FUNCTION_BLOCK FB_Machine
VAR_INPUT
	// ========================== SEPARATING MODULE =======================================
	// Separating module - clamp cylinder
	bSeparatingClampDiag						:		BOOL	:=	FALSE;
	bSeparatingClampTemp						:		BOOL	:=	TRUE;
	bSeparatingClampRecord						:		BOOL	:=	TRUE;
	// Separating module - barrier cylinder
	bSeparatingBarrierDiag						:		BOOL	:=	TRUE;
	bSeparatingBarrierTemp						:		BOOL	:=	TRUE;
	bSeparatingBarrierRecord					:		BOOL	:=	FALSE;
	// ========================== SORTING MODULES ==========================================
	bMetalSortingCylinderDiag					:		BOOL	:= 	TRUE;
	bMetalSortingCylinderTemp					:		BOOL	:=	FALSE;
	bMetalSortingCylinderRecord					:		BOOL	:=	FALSE;
	
	bPlasticSortingCylinderDiag					:		BOOL	:=	FALSE;
	bPlasticSortingCylinderTemp					:		BOOL	:=	FALSE;
	bPlasticSortingCylinderRecord				:		BOOL	:=	FALSE;
END_VAR
VAR
	// ============================= ERROR ==================================================
	bError										:		BOOL;
	// ========================== Axis Variable =============================================
	fAxisVelo									:		LREAL;
	fAxisVeloLastCycle							:		LREAL;
	// ======================== State machine variables =====================================
	bStarted									:		BOOL;
	bStopped									:		BOOL;
	bReset								AT %Q* 	: 		BOOL;
	bAborted									:		BOOL;
	bIdle										:		BOOL;
	bAuto										:		BOOL;
	bSemi										:		BOOL;
	bManual										:		BOOL;
	bMaintenance								:		BOOL;
	// ========================== Machine submodules ========================================
	fbSeparatingModule							:		FB_SeparatingModule;
	fbMetalSortingModule						:		FB_SortingModule;
	fbPlasticSortingModule						:		FB_SortingModule;
	fbComprAir									:		FB_SignalHandlingIntern;
	fbPowerSupply								:		FB_SignalHandlingIntern;
	// Visualization
	// ========================== Buttons ========================================
	fbButtonStart								:		FB_SignalHandlingIntern;
	fbButtonStop								:		FB_SignalHandlingIntern;
	fbButtonReset								:		FB_SignalHandlingIntern;
	fbButtonAbort								:		FB_SignalHandlingIntern;
	fbButtonAuto								:		FB_SignalHandlingIntern;
	fbButtonSemi								:		FB_SignalHandlingIntern;
	fbButtonManual								:		FB_SignalHandlingIntern;
	fbButtonMaintenance							:		FB_SignalHandlingIntern;
	fbButtonComprAir							:		FB_SignalHandlingIntern;
	fbButtonPower								:		FB_SignalHandlingIntern;
	// ========================== State machine ==================================
	fbStateMachineAuto							:		PS_PackML_StateMachine_Auto;
	fbStateMachineSemiAuto						:		PS_PackML_StateMachine_SemiAuto;
	fbStateMachineManual						:		PS_PackML_StateMachine_Manual;
	fbStateMachineMaintenance					:		PS_PackML_StateMachine_Maintenance;
	
	e_PMLState									:		E_PMLState			:=	E_PMLState.IDLE;
	e_PMLStateRequest							:		E_PMLState;
	e_PMLUnitMode								:		E_PMLUnitMode		:=	E_PMLUnitMode.IDLE;
	e_PMLUnitModeRequest						:		E_PMLUnitMode;
		fbUnitModeManager						:		PS_PackML_UnitModeManager;
	// ======================= Common variables ===================================
	bInit										:		BOOL;
	bAxisEnable									:		BOOL;
	bManualAxisEnable							:		BOOL;
	
	fbTriggerStartButton						:		R_TRIG;
	fbTriggerSeparated							:		R_TRIG;
	fbTriggerMetalSorted						:		R_TRIG;
	fbTriggerPlasticSorted						:		R_TRIG;
	
	nBoxesOnTransport							:		UINT;
	
	aClampTemps									:		ARRAY [1..100] OF LREAL;
	aBarrierTemps								:		ARRAY [1..100] OF LREAL;
	aMetalCylTemps								:		ARRAY [1..100] OF LREAL;
	aPlasticCylTemps							:		ARRAY [1..100] OF LREAL;
	
	bStartingIsSetToTrue						:		BOOL;
	bResetIsSetToTrue							:		BOOL;
	bHaltIsSetToTrue							:		BOOL;
END_VAR
VAR CONSTANT
	// ======================= Axis parameters ===================================
	cAxisVeloAutomatic							:		LREAL	:=		100.0;
	cAxisVeloNonAutomatic						:		LREAL	:=		50.0;
	// =============== Separating module parameters ===============================
	tSeparatingTimeOutClamp						:		TIME	:=		T#4S;
	tSeparatingRecordIntervalClamp				:		TIME	:=		T#1S;
	
	tSeparatingTimeOutBarrier					:		TIME	:=		T#3S;
	tSeparatingRecordIntervalBarrier			:		TIME	:=		T#1S;
	tSeparatingTimeBarrierAtWork				:		TIME	:=		T#3.5S;
	
	rSeparatingClampTempMin						:		LREAL	:=		5.0;
	rSeparatingClampTempMax						:		LREAL	:=		78.0;
	rSeparatingBarrierTempMin					:		LREAL	:= 		2.0;
	rSeparatingBarrierTempMax					:		LREAL	:= 		95.0;
	// =============== Sorting module parameters ==================================
	tSortingMetalTimeOutCyl						:		TIME	:=		T#3S;
	tSortingMetalRecordIntervalCyl				:		TIME	:=		T#1S;
	tSortingMetalSensorDelay					:		TIME	:=		T#2S;
	tSortingMetalMoveAxisDelay					:		TIME	:=		T#3S;

	rSortingMetalCylTempMin						:		LREAL	:= 		2.0;
	rSortingMetalCylTempMax						:		LREAL	:= 		95.0;
	
	tSortingPlasticTimeOutCyl					:		TIME	:=		T#3S;
	tSortingPlasticRecordIntervalCyl			:		TIME	:=		T#1S;
	tSortingPlasticSensorDelay					:		TIME	:=		T#2S;
	tSortingPlasticMoveAxisDelay				:		TIME	:=		T#3S;
	
	rSortingPlasticCylTempMin					:		LREAL	:= 		2.0;
	rSortingPlasticCylTempMax					:		LREAL	:= 		95.0;
END_VAR


	// Modules errors
	bError	:=	fbSeparatingModule.bAxisError OR fbSeparatingModule.bBarrierError OR fbSeparatingModule.bClampError OR
				fbMetalSortingModule.bAxisError OR fbMetalSortingModule.bCylError OR
				fbPlasticSortingModule.bAxisError OR fbPlasticSortingModule.bCylError;
				
	// Axis velocity
	IF (e_PMLUnitMode = E_PMLUnitMode.AUTOMATIC OR e_PMLUnitMode = E_PMLUnitMode.SEMIAUTOMATIC) THEN
		fAxisVelo		:=		cAxisVeloAutomatic;
	ELSE
		fAxisVelo		:=		cAxisVeloNonAutomatic;	
	END_IF
 
	// Separeted and sorted boxes output transfer
	fbTriggerSeparated(		CLK		:=		fbSeparatingModule.bSeparated);
	fbTriggerMetalSorted(	CLK		:=		fbMetalSortingModule.bSorted);
	fbTriggerPlasticSorted(	CLK		:=		fbPlasticSortingModule.bSorted);
	
	// Temperatures of modules
	aBarrierTemps					:=		fbSeparatingModule.aBarrierTemp;
	aClampTemps						:=		fbSeparatingModule.aClampTemp;
	aMetalCylTemps					:=		fbMetalSortingModule.aCylTemps;
	aPlasticCylTemps				:=		fbPlasticSortingModule.aCylTemps;
	
	// Cylinder options of modules
	fbSeparatingModule.CylinderOptions(		bClampDiag			:=				bSeparatingClampDiag,
											bClampTemp			:=				bSeparatingClampTemp,
											bClampRecord		:=				bSeparatingClampRecord,
											bBarrierDiag		:=				bSeparatingBarrierDiag,
											bBarrierTemp		:=				bSeparatingBarrierTemp,
											bBarrierRecord		:=				bSeparatingBarrierRecord);
											
	fbMetalSortingModule.CylinderOptions(	bCylDiag			:=				bMetalSortingCylinderDiag,
											bCylTemp			:=				bMetalSortingCylinderTemp,
											bCylRecord			:=				bMetalSortingCylinderRecord);
											
	fbPlasticSortingModule.CylinderOptions(	bCylDiag			:=				bPlasticSortingCylinderDiag,
											bCylTemp			:=				bPlasticSortingCylinderTemp,
											bCylRecord			:=				bPlasticSortingCylinderRecord);
											
	General_Init();
	
	General_Enable();
	
	General_ModuleInputs();
	
	General_SetOutputs();
	
	General_Requests();
	
	General_StateMachine();

METHOD PRIVATE General_Enable
VAR_INPUT
END_VAR

	// Power supply
	fbPowerSupply.Enable(	bEnable					:=		TRUE);
	fbButtonPower.Enable(	bEnable					:=		TRUE);
	
	
	fbPowerSupply.bInputSignal					:=		fbButtonPower.bOutputSignal;
	
	// Axis control
	IF (e_PMLState	:=	E_PMLState.ABORTED) THEN
		bAxisEnable				:=		FALSE;
	ELSIF fbPowerSupply.bOutputSignal THEN
		bAxisEnable				:=		TRUE;		
	END_IF
	
	bManualAxisEnable	:=	fbPowerSupply.bOutputSignal AND (e_PMLState	:=	E_PMLState.EXECUTE) AND (e_PMLUnitMode = E_PMLUnitMode.MANUAL OR e_PMLUnitMode = E_PMLUnitMode.MAINTENANCE);
	
	// Compressed air control
	IF NOT (e_PMLUnitMode		:=		E_PMLUnitMode.MAINTENANCE) THEN
		fbComprAir				:=		fbPowerSupply.bOutputSignal;
	ELSE
		fbComprAir				:=		fbButtonComprAir;
	END_IF
	
	fbComprAir.Enable(			bEnable		:=		TRUE);
	fbButtonComprAir.Enable(	bEnable		:=		(e_PMLUnitMode = E_PMLUnitMode.MAINTENANCE));
	
	// Separating module 
	fbSeparatingModule.Enable(		bAxisEnable				:=			bAxisEnable,
									bComprAirEnable			:=			fbComprAir.bOutputSignal OR fbButtonComprAir.bOutputSignal,
									bManualAxisEnable		:=			bManualAxisEnable,
									bSensorEnable			:=			TRUE);
								
	// Sorting plastic
	fbPlasticSortingModule.Enable(	bAxisEnable				:=			bAxisEnable,
									bComprAirEnable			:=			fbComprAir.bOutputSignal OR fbButtonComprAir.bOutputSignal,
									bManualAxisEnable		:=			bManualAxisEnable,
									bSensorEnable			:=			TRUE);
	
	// Sorting metal
	fbMetalSortingModule.Enable(	bAxisEnable				:=			bAxisEnable,
									bComprAirEnable			:=			fbComprAir.bOutputSignal OR fbButtonComprAir.bOutputSignal,
									bManualAxisEnable		:=			bManualAxisEnable,
									bSensorEnable			:=			TRUE);
									
	// States
	fbButtonStart.Enable		(	bEnable					:=			NOT bError);
	
	fbButtonStop.Enable			(	bEnable					:=			((e_PMLState = E_PMLState.STOPPING) OR (e_PMLState = E_PMLState.EXECUTE) OR (e_PMLState = E_PMLState.IDLE)));
	
	fbButtonAbort.bInputSignal								:=			fbPowerSupply.bOutputSignal;
	fbButtonAbort.Enable		(	bEnable					:=			((e_PMLState = E_PMLState.ABORTING) OR (e_PMLState = E_PMLState.STOPPING) OR (e_PMLState = E_PMLState.EXECUTE) OR (e_PMLState = E_PMLState.RESETTING)));
	
	fbButtonReset.Enable		(	bEnable					:=			(e_PMLState = E_PMLState.STOPPED)); 
	
	// Unit Modes
	fbButtonAuto.Enable			(	bEnable					:=			((e_PMLState = E_PMLState.IDLE) AND (e_PMLUnitMode <> E_PMLUnitMode.AUTOMATIC)));
	
	fbButtonSemi.Enable			(	bEnable					:=			((e_PMLState = E_PMLState.IDLE) AND (e_PMLUnitMode <> E_PMLUnitMode.SEMIAUTOMATIC)));
	
	fbButtonManual.Enable		(	bEnable					:=			((e_PMLState = E_PMLState.IDLE) AND (e_PMLUnitMode <> E_PMLUnitMode.MANUAL)));
	
	fbButtonMaintenance.Enable	(	bEnable					:=			((e_PMLState = E_PMLState.IDLE) AND (e_PMLUnitMode <> E_PMLUnitMode.MAINTENANCE)));
END_METHOD

METHOD PRIVATE General_Init
VAR_INPUT
END_VAR

	IF NOT bInit THEN
	// ================================ Separating module parameters ==========================================
		// Clamp cylinder
		fbSeparatingModule.tProp_TimeIntervalClamp				:=		tSeparatingRecordIntervalClamp;
		fbSeparatingModule.tProp_TimeOutClamp					:=		tSeparatingTimeOutClamp;
		
		fbSeparatingModule.nProp_TempMaxClamp					:=		rSeparatingClampTempMax;
		fbSeparatingModule.nProp_TempMinClamp					:=		rSeparatingClampTempMin;
				
		// Barrier cylinder
		fbSeparatingModule.tProp_TimeIntervalBarrier			:=		tSeparatingRecordIntervalBarrier;
		fbSeparatingModule.tProp_TimeOutBarrier					:=		tSeparatingTimeOutBarrier;
		
		fbSeparatingModule.tBarrierAtWorkPos					:=		tSeparatingTimeBarrierAtWork;
		
		fbSeparatingModule.nProp_TempMaxBarrier					:=		rSeparatingBarrierTempMax;
		fbSeparatingModule.nProp_TempMinBarrier					:=		rSeparatingBarrierTempMin;
	

	// ============================== Sorting metal module parameters ==========================================
		fbMetalSortingModule.tProp_AxisMoving					:=		tSortingMetalMoveAxisDelay;
		fbMetalSortingModule.tProp_CylRecInterval				:=		tSortingMetalRecordIntervalCyl;
		fbMetalSortingModule.tProp_CylTimeOut					:=		tSortingMetalTimeOutCyl;
		fbMetalSortingModule.tProp_SensorDelay					:=		tSortingMetalSensorDelay;
		
		fbMetalSortingModule.nProp_CylTempMax					:=		rSortingMetalCylTempMax;
		fbMetalSortingModule.nProp_CylTempMin					:=		rSortingMetalCylTempMin;
			
	// ============================== Sorting plastic module parameters ==========================================
		fbPlasticSortingModule.tProp_AxisMoving					:=		tSortingPlasticMoveAxisDelay;
		fbPlasticSortingModule.tProp_CylRecInterval				:=		tSortingPlasticRecordIntervalCyl;
		fbPlasticSortingModule.tProp_CylTimeOut					:=		tSortingPlasticTimeOutCyl;
		fbPlasticSortingModule.tProp_SensorDelay				:=		tSortingPlasticSensorDelay;
		
		fbPlasticSortingModule.nProp_CylTempMax					:=		rSortingPlasticCylTempMax;
		fbPlasticSortingModule.nProp_CylTempMin					:=		rSortingPlasticCylTempMin;
		
		bInit			:=		TRUE;
	END_IF
END_METHOD

METHOD PRIVATE General_ModuleInputs
VAR_INPUT
END_VAR

	// Separating module
		fbSeparatingModule.bExecute								:=		(e_PMLState :=	E_PMLState.EXECUTE);
		
		// Axis velocity has changed
		IF (fAxisVeloLastCycle <> fAxisVelo) THEN
			fbSeparatingModule.fAxisVelocity					:=		fAxisVelo;
		END_IF
	
			fbSeparatingModule.nBoxOnConveyor					:=		nBoxesOnTransport;
	// Sorting module plastic
		// Axis velocity has changed
		IF (fAxisVeloLastCycle <> fAxisVelo) THEN
			fbPlasticSortingModule.fAxisVelocity				:=		fAxisVelo;
		END_IF
	
	// Sorting module metal
		// Axis velocity has changed
		IF (fAxisVeloLastCycle <> fAxisVelo) THEN
			fbMetalSortingModule.fAxisVelocity				:=		fAxisVelo;
		END_IF
	
		// Save axis velocity of actual cycle for the next cycle
		fAxisVeloLastCycle			:=			fAxisVelo;
END_METHOD

METHOD PRIVATE General_Requests
VAR_INPUT
END_VAR

	// State requests
	fbTriggerStartButton(CLK	:=		fbButtonStart);
	
	IF fbTriggerStartButton.Q THEN
		IF e_PMLState = E_PMLState.ABORTED THEN
			e_PMLStateRequest	:=	E_PMLState.CLEARING;
			
		ELSIF e_PMLState 	= E_PMLState.STOPPED THEN
			e_PMLStateRequest	:=	E_PMLState.RESETTING;
			
		ELSIF e_PMLState	=	E_PMLState.IDLE AND fbPowerSupply.bOutputSignal THEN
			e_PMLStateRequest	:=	E_PMLState.STARTING;
		END_IF
	ELSIF  fbButtonStop THEN
		e_PMLStateRequest	:=	E_PMLState.STOPPING;
	
	ELSIF	fbButtonReset THEN
		e_PMLStateRequest	:=	E_PMLState.RESETTING;
	END_IF
	
	// Mode requests
	IF fbButtonAuto.bOutputSignal THEN
		e_PMLUnitModeRequest	:=		E_PMLUnitMode.AUTOMATIC;
	ELSIF fbButtonSemi.bOutputSignal THEN
		e_PMLUnitModeRequest	:=		E_PMLUnitMode.SEMIAUTOMATIC;
	ELSIF fbButtonManual.bOutputSignal THEN
		e_PMLUnitModeRequest	:=		E_PMLUnitMode.MANUAL;
	ELSIF fbButtonMaintenance.bOutputSignal THEN
		e_PMLUnitModeRequest	:=		E_PMLUnitMode.MAINTENANCE;
	END_IF
	
	// UnitModeManager call
	IF fbButtonAuto.bOutputSignal OR fbButtonSemi.bOutputSignal OR fbButtonManual.bOutputSignal OR fbButtonMaintenance.bOutputSignal THEN
		fbUnitModeManager(	bExecute					:=		TRUE,
							ePMLUnitModeCommand			:=		e_PMLUnitModeRequest,
							ePMLState					:=		e_PMLState);
	END_IF
	
	IF fbUnitModeManager.bDone THEN
		e_PMLUnitMode	:=		fbUnitModeManager.ePMLUnitModeStatus;
		
		fbUnitModeManager(	bExecute					:=		FALSE);
	END_IF
END_METHOD

METHOD PRIVATE General_SetOutputs
VAR_INPUT
END_VAR

	// State variables
	bStarted								:=			(e_PMLState = E_PMLState.EXECUTE);
	bStopped								:=			(e_PMLState = E_PMLState.STOPPED);
	bReset									:=			(e_PMLState = E_PMLState.RESETTING);
	bAborted								:=			(e_PMLState = E_PMLState.ABORTED);
	bIdle									:=			(e_PMLState = E_PMLState.IDLE);
	
	// Unit Mode variables
	bAuto									:=			(e_PMLUnitMode = E_PMLUnitMode.AUTOMATIC);
	bSemi									:=			(e_PMLUnitMode = E_PMLUnitMode.SEMIAUTOMATIC);
	bManual									:=			(e_PMLUnitMode = E_PMLUnitMode.MANUAL);
	bMaintenance							:=			(e_PMLUnitMode = E_PMLUnitMode.MAINTENANCE);
	
	// Power supply and air
	fbPowerSupply.SetOutput();
	fbComprAir.SetOutput();
	
	// Subsystems
	fbSeparatingModule.InputOutput();
	fbPlasticSortingModule.InputOutput();
	fbMetalSortingModule.InputOutput();
	
	// ======================= Buttons =========================================================================
		// Power supply and air
		fbButtonPower.SetOutput();
		fbButtonComprAir.SetOutput();
			
		// States
		fbButtonStart.SetOutput();
		fbButtonStop.SetOutput();
		fbButtonReset.SetOutput();
		fbButtonAbort.SetOutput();
		
		// Modes
		fbButtonAuto.SetOutput();
		fbButtonSemi.SetOutput();
		fbButtonManual.SetOutput();
		fbButtonMaintenance.SetOutput();
END_METHOD

METHOD PRIVATE General_StateMachine
VAR_INPUT
END_VAR

	// Mode and State Handling
	CASE e_PMLUnitMode OF
		E_PMLUnitMode.AUTOMATIC:
			fbStateMachineAuto(			Start		:=			e_PMLStateRequest = E_PMLState.STARTING,
										Stop		:=			fbButtonStop.bOutputSignal,
										Reset		:=			e_PMLStateRequest = E_PMLState.RESETTING OR fbButtonReset.bOutputSignal,
										Clear		:=			e_PMLStateRequest = E_PMLState.CLEARING,
										Abort		:=			e_PMLStateRequest = E_PMLState.ABORTING OR (bError AND e_PMLStateRequest = E_PMLState.EXECUTE));
								
					e_PMLState		:=			fbStateMachineAuto.ePMLState;
					
					// State internal commands handling + StateComplete signal for switching PackML_StateMachine
					Operating_Automatic();
					
		E_PMLUnitMode.SEMIAUTOMATIC:
			fbStateMachineSemiAuto(		Start		:=			e_PMLStateRequest = E_PMLState.STARTING,
										Stop		:=			fbButtonStop.bOutputSignal,
										Reset		:=			e_PMLStateRequest = E_PMLState.RESETTING OR fbButtonReset.bOutputSignal,
										Clear		:=			e_PMLStateRequest = E_PMLState.CLEARING,
										Abort		:=			e_PMLStateRequest = E_PMLState.ABORTING OR (bError AND e_PMLStateRequest = E_PMLState.EXECUTE));
								
					e_PMLState		:=			fbStateMachineSemiAuto.ePMLState;
		
					// State internal commands handling + StateComplete signal for switching PackML_StateMachine
					Operating_SemiAutomatic();
					
		E_PMLUnitMode.MANUAL:
			fbStateMachineManual(		Start		:=			e_PMLStateRequest = E_PMLState.STARTING,
										Stop		:=			fbButtonStop.bOutputSignal,
										Reset		:=			e_PMLStateRequest = E_PMLState.RESETTING OR fbButtonReset.bOutputSignal,
										Clear		:=			e_PMLStateRequest = E_PMLState.CLEARING,
										Abort		:=			e_PMLStateRequest = E_PMLState.ABORTING OR (bError AND e_PMLStateRequest = E_PMLState.EXECUTE));
								
					e_PMLState		:=			fbStateMachineManual.ePMLState;

					// State internal commands handling + StateComplete signal for switching PackML_StateMachine
					Operating_Manual();
					
		E_PMLUnitMode.MAINTENANCE:
			fbStateMachineMaintenance(	Start		:=			e_PMLStateRequest = E_PMLState.STARTING,
										Stop		:=			fbButtonStop.bOutputSignal,
										Reset		:=			e_PMLStateRequest = E_PMLState.RESETTING OR fbButtonReset.bOutputSignal,
										Clear		:=			e_PMLStateRequest = E_PMLState.CLEARING,
										Abort		:=			e_PMLStateRequest = E_PMLState.ABORTING OR (bError AND e_PMLStateRequest = E_PMLState.EXECUTE));
								
					e_PMLState		:=			fbStateMachineMaintenance.ePMLState;
					
					// State internal commands handling + StateComplete signal for switching PackML_StateMachine
					Operating_Maintenance();		
	END_CASE
END_METHOD

METHOD PRIVATE Operating_Automatic
VAR_INPUT
END_VAR

	CASE e_PMLState OF
		
		E_PMLState.IDLE:
			IF bResetIsSetToTrue THEN
				bResetIsSetToTrue		:=	FALSE;
				fbSeparatingModule.Reset(		bReset		:=	FALSE);
				fbMetalSortingModule.Reset(		bReset		:=	FALSE);
				fbPlasticSortingModule.Reset(	bReset		:=	FALSE);

				THIS^.fbStateMachineAuto.StateComplete		:=	FALSE;	
			END_IF
			
		E_PMLState.STARTING:
			IF NOT bStartingIsSetToTrue THEN
				bStartingIsSetToTrue	:=	TRUE;
				fbSeparatingModule.Starting(	bStarting	:=	TRUE);
				fbMetalSortingModule.Starting(	bStarting	:=	TRUE);
				fbPlasticSortingModule.Starting(bStarting	:=	TRUE);
			END_IF	
			
			IF fbSeparatingModule.bState_StartingDone AND fbMetalSortingModule.bState_StartingDone AND fbPlasticSortingModule.bState_StartingDone THEN
					THIS^.fbStateMachineAuto.StateComplete		:=	TRUE;
			END_IF
			
		E_PMLState.EXECUTE:
			IF bStartingIsSetToTrue THEN
				bStartingIsSetToTrue	:=	FALSE;
				fbSeparatingModule.Starting(	bStarting	:=	FALSE);
				fbMetalSortingModule.Starting(	bStarting	:=	FALSE);
				fbPlasticSortingModule.Starting(bStarting	:=	FALSE);
				
				THIS^.fbStateMachineAuto.StateComplete		:=	FALSE;
			END_IF
 			
				fbSeparatingModule.Automatic();
				fbMetalSortingModule.Automatic();
				fbPlasticSortingModule.Automatic();
				
				IF fbTriggerSeparated.Q THEN
					nBoxesOnTransport	:=	nBoxesOnTransport + 1;
				END_IF
				
				IF fbTriggerMetalSorted.Q THEN
					nBoxesOnTransport	:=	nBoxesOnTransport - 1;
				END_IF
				
				IF fbTriggerPlasticSorted.Q THEN
					nBoxesOnTransport	:=	nBoxesOnTransport - 1;
				END_IF

		E_PMLState.ABORTING:
				IF NOT bHaltIsSetToTrue THEN
					bHaltIsSetToTrue	:=	TRUE;
					fbSeparatingModule.Stop(		bStop		:=	TRUE);
					fbMetalSortingModule.Stop(		bStop		:=	TRUE);
					fbPlasticSortingModule.Stop(	bStop		:=	TRUE);
				END_IF
				
				IF fbSeparatingModule.bState_HaltDone AND fbMetalSortingModule.bState_HaltDone AND fbPlasticSortingModule.bState_HaltDone THEN
					THIS^.fbStateMachineAuto.StateComplete		:=	TRUE;
				END_IF
			
		E_PMLState.ABORTED:
				IF bHaltIsSetToTrue THEN
					bHaltIsSetToTrue	:=	FALSE;
					fbSeparatingModule.Stop(		bStop		:=	FALSE);
					fbMetalSortingModule.Stop(		bStop		:=	FALSE);
					fbPlasticSortingModule.Stop(	bStop		:=	FALSE);
				END_IF
				
				IF THIS^.fbStateMachineAuto.StateComplete THEN
					THIS^.fbStateMachineAuto.StateComplete		:=	FALSE;
				END_IF
				
		E_PMLState.CLEARING:
				THIS^.fbStateMachineAuto.StateComplete		:=	TRUE;
				
		E_PMLState.STOPPING:
				IF fbTriggerSeparated.Q THEN
					nBoxesOnTransport	:=	nBoxesOnTransport	+	1;
				END_IF

				IF fbTriggerMetalSorted.Q THEN
					nBoxesOnTransport	:=	nBoxesOnTransport	-	1;
				END_IF

				IF fbTriggerPlasticSorted.Q THEN
					nBoxesOnTransport	:=	nBoxesOnTransport	-	1;
				END_IF

				IF nBoxesOnTransport = 0 AND NOT bHaltIsSetToTrue THEN
					bHaltIsSetToTrue	:=	TRUE;
					fbSeparatingModule.Stop(	bStop		:=		TRUE);
					fbMetalSortingModule.Stop(	bStop		:=		TRUE);
					fbPlasticSortingModule.Stop(bStop		:=		TRUE);
				END_IF
				
				IF fbSeparatingModule.bState_HaltDone AND fbMetalSortingModule.bState_HaltDone AND fbPlasticSortingModule.bState_HaltDone AND nBoxesOnTransport = 0 THEN
					THIS^.fbStateMachineAuto.StateComplete	:=	TRUE;
				END_IF
							
		E_PMLState.STOPPED:
				IF bHaltIsSetToTrue THEN
					bHaltIsSetToTrue	:=	FALSE;
					fbSeparatingModule.Stop(	bStop		:=		FALSE);
					fbMetalSortingModule.Stop(	bStop		:=		FALSE);
					fbPlasticSortingModule.Stop(bStop		:=		FALSE);
				END_IF
				
				IF THIS^.fbStateMachineAuto.StateComplete THEN
					THIS^.fbStateMachineAuto.StateComplete	:=		FALSE;
				END_IF
								
		E_PMLState.RESETTING:
				IF NOT bResetIsSetToTrue THEN
					bResetIsSetToTrue 	:=	TRUE;
					
					fbSeparatingModule.Reset(	bReset		:=		TRUE);
					fbMetalSortingModule.Reset(	bReset		:=		TRUE);
					fbPlasticSortingModule.Reset(bReset 	:=		TRUE);
				END_IF
				
				IF fbSeparatingModule.bState_ResetDone AND fbMetalSortingModule.bState_ResetDone AND fbPlasticSortingModule.bState_ResetDone AND
					fbSeparatingModule.bState_BarrierAtBasePos AND fbSeparatingModule.bState_ClampAtBasePos AND fbMetalSortingModule.bState_CylAtBasePos AND fbPlasticSortingModule.bState_CylAtBasePos THEN
					nBoxesOnTransport					:=	0;
					fbStateMachineAuto.StateComplete	:=	TRUE;
				END_IF
	END_CASE
END_METHOD

METHOD PRIVATE Operating_Maintenance
VAR_INPUT
END_VAR

	CASE e_PMLState OF
		
		E_PMLState.IDLE:
			IF bResetIsSetToTrue THEN
				bResetIsSetToTrue		:=		FALSE;
				fbSeparatingModule.Reset(		bReset			:=		FALSE);
				fbMetalSortingModule.Reset(		bReset			:=		FALSE);
				fbPlasticSortingModule.Reset(	bReset			:=		FALSE);
			
				THIS^.fbStateMachineMaintenance.StateComplete		:=		FALSE;
			END_IF
		
		E_PMLState.STARTING:
			IF NOT bStartingIsSetToTrue THEN
				bStartingIsSetToTrue	:=		TRUE;
				fbSeparatingModule.Starting(	bStarting		:=		TRUE);
				fbMetalSortingModule.Starting(	bStarting		:=		TRUE);
				fbPlasticSortingModule.Starting(bStarting		:=		TRUE);
			END_IF
			
			IF fbSeparatingModule.bState_StartingDone AND fbMetalSortingModule.bState_StartingDone AND fbPlasticSortingModule.bState_StartingDone THEN
				THIS^.fbStateMachineMaintenance.StateComplete		:=		TRUE;
			END_IF		
		
		E_PMLState.EXECUTE:
			IF bStartingIsSetToTrue	THEN
				bStartingIsSetToTrue	:=	FALSE;
				fbSeparatingModule.Starting(	bStarting		:=		FALSE);
				fbMetalSortingModule.Starting(	bStarting		:=		FALSE);
				fbPlasticSortingModule.Starting(bStarting		:=		FALSE);
				
				THIS^.fbStateMachineMaintenance.StateComplete		:=		FALSE;
			END_IF
				
				fbSeparatingModule.Maintain();
				fbMetalSortingModule.Maintenance();
				fbPlasticSortingModule.Maintenance();
				
		E_PMLState.ABORTING:
			IF NOT bHaltIsSetToTrue THEN
				bHaltIsSetToTrue		:=	TRUE;
				fbSeparatingModule.Stop(		bStop 			:= 		TRUE);
				fbMetalSortingModule.Stop(		bStop 			:= 		TRUE);
				fbPlasticSortingModule.Stop(	bStop 			:=		TRUE);
			END_IF
			
			IF fbSeparatingModule.bState_HaltDone AND fbMetalSortingModule.bState_HaltDone AND fbPlasticSortingModule.bState_HaltDone THEN
				THIS^.fbStateMachineMaintenance.StateComplete		:=		TRUE;
			END_IF
		
		E_PMLState.ABORTED:
			IF bHaltIsSetToTrue	THEN
				bHaltIsSetToTrue		:=	FALSE;
				fbSeparatingModule.Stop(		bStop 			:= 		FALSE);
				fbMetalSortingModule.Stop(		bStop 			:= 		FALSE);
				fbPlasticSortingModule.Stop(	bStop 			:=		FALSE);
			END_IF
			
			IF THIS^.fbStateMachineMaintenance.StateComplete THEN
				THIS^.fbStateMachineMaintenance.StateComplete		:=		FALSE;
			END_IF
			
		E_PMLState.CLEARING:
			
			THIS^.fbStateMachineMaintenance.StateComplete			:=		TRUE;
		
		E_PMLState.STOPPING:
			IF NOT bHaltIsSetToTrue THEN
				bHaltIsSetToTrue		:=	TRUE;
				fbSeparatingModule.Stop(		bStop 			:= 		TRUE);
				fbMetalSortingModule.Stop(		bStop 			:= 		TRUE);
				fbPlasticSortingModule.Stop(	bStop 			:=		TRUE);
			END_IF
			
			IF fbSeparatingModule.bState_HaltDone AND fbMetalSortingModule.bState_HaltDone AND fbPlasticSortingModule.bState_HaltDone THEN
				THIS^.fbStateMachineMaintenance.StateComplete		:=		TRUE;
			END_IF
		
		E_PMLState.STOPPED:
			IF bHaltIsSetToTrue	THEN
				bHaltIsSetToTrue		:=	FALSE;
				fbSeparatingModule.Stop(		bStop 			:= 		FALSE);
				fbMetalSortingModule.Stop(		bStop 			:= 		FALSE);
				fbPlasticSortingModule.Stop(	bStop 			:=		FALSE);
			END_IF
			
			IF THIS^.fbStateMachineMaintenance.StateComplete THEN
				THIS^.fbStateMachineMaintenance.StateComplete		:=		FALSE;
			END_IF
			
		E_PMLState.RESETTING:
		
			IF NOT bResetIsSetToTrue THEN
				bResetIsSetToTrue		:=	TRUE;
				fbSeparatingModule.Reset(	bReset		:=		TRUE);
				fbMetalSortingModule.Reset(	bReset		:=		TRUE);
				fbPlasticSortingModule.Reset(bReset 	:=		TRUE);
			END_IF
				
			IF fbSeparatingModule.bState_ResetDone AND fbMetalSortingModule.bState_ResetDone AND fbPlasticSortingModule.bState_ResetDone AND
				fbSeparatingModule.bState_BarrierAtBasePos AND fbSeparatingModule.bState_ClampAtBasePos AND fbMetalSortingModule.bState_CylAtBasePos AND fbPlasticSortingModule.bState_CylAtBasePos THEN
					nBoxesOnTransport					:=	0;
					fbStateMachineMaintenance.StateComplete	:=	TRUE;
			END_IF
	END_CASE
END_METHOD

METHOD PRIVATE Operating_Manual
VAR_INPUT
END_VAR

	CASE e_PMLState OF
		
		E_PMLState.IDLE:
			IF bResetIsSetToTrue THEN
				bResetIsSetToTrue		:=		FALSE;
				fbSeparatingModule.Reset(		bReset			:=		FALSE);
				fbMetalSortingModule.Reset(		bReset			:=		FALSE);
				fbPlasticSortingModule.Reset(	bReset			:=		FALSE);
			
				THIS^.fbStateMachineManual.StateComplete		:=		FALSE;
			END_IF
		
		E_PMLState.STARTING:
			IF NOT bStartingIsSetToTrue THEN
				bStartingIsSetToTrue	:=		TRUE;
				fbSeparatingModule.Starting(	bStarting		:=		TRUE);
				fbMetalSortingModule.Starting(	bStarting		:=		TRUE);
				fbPlasticSortingModule.Starting(bStarting		:=		TRUE);
			END_IF
			
			IF fbSeparatingModule.bState_StartingDone AND fbMetalSortingModule.bState_StartingDone AND fbPlasticSortingModule.bState_StartingDone THEN
				THIS^.fbStateMachineManual.StateComplete		:=		TRUE;
			END_IF		
		
		E_PMLState.EXECUTE:
			IF bStartingIsSetToTrue	THEN
				bStartingIsSetToTrue	:=	FALSE;
				fbSeparatingModule.Starting(	bStarting		:=		FALSE);
				fbMetalSortingModule.Starting(	bStarting		:=		FALSE);
				fbPlasticSortingModule.Starting(bStarting		:=		FALSE);
				
				THIS^.fbStateMachineManual.StateComplete		:=		FALSE;
			END_IF
				
				fbSeparatingModule.Manual();
				fbMetalSortingModule.Manual();
				fbPlasticSortingModule.Manual();
				
		E_PMLState.ABORTING:
			IF NOT bHaltIsSetToTrue THEN
				bHaltIsSetToTrue		:=	TRUE;
				fbSeparatingModule.Stop(		bStop 			:= 		TRUE);
				fbMetalSortingModule.Stop(		bStop 			:= 		TRUE);
				fbPlasticSortingModule.Stop(	bStop 			:=		TRUE);
			END_IF
			
			IF fbSeparatingModule.bState_HaltDone AND fbMetalSortingModule.bState_HaltDone AND fbPlasticSortingModule.bState_HaltDone THEN
				THIS^.fbStateMachineManual.StateComplete		:=		TRUE;
			END_IF
		
		E_PMLState.ABORTED:
			IF bHaltIsSetToTrue	THEN
				bHaltIsSetToTrue		:=	FALSE;
				fbSeparatingModule.Stop(		bStop 			:= 		FALSE);
				fbMetalSortingModule.Stop(		bStop 			:= 		FALSE);
				fbPlasticSortingModule.Stop(	bStop 			:=		FALSE);
			END_IF
			
			IF THIS^.fbStateMachineManual.StateComplete THEN
				THIS^.fbStateMachineManual.StateComplete		:=		FALSE;
			END_IF
			
		E_PMLState.CLEARING:
			
			THIS^.fbStateMachineManual.StateComplete			:=		TRUE;
		
		E_PMLState.STOPPING:
			IF NOT bHaltIsSetToTrue THEN
				bHaltIsSetToTrue		:=	TRUE;
				fbSeparatingModule.Stop(		bStop 			:= 		TRUE);
				fbMetalSortingModule.Stop(		bStop 			:= 		TRUE);
				fbPlasticSortingModule.Stop(	bStop 			:=		TRUE);
			END_IF
			
			IF fbSeparatingModule.bState_HaltDone AND fbMetalSortingModule.bState_HaltDone AND fbPlasticSortingModule.bState_HaltDone THEN
				THIS^.fbStateMachineManual.StateComplete		:=		TRUE;
			END_IF
		
		E_PMLState.STOPPED:
			IF bHaltIsSetToTrue	THEN
				bHaltIsSetToTrue		:=	FALSE;
				fbSeparatingModule.Stop(		bStop 			:= 		FALSE);
				fbMetalSortingModule.Stop(		bStop 			:= 		FALSE);
				fbPlasticSortingModule.Stop(	bStop 			:=		FALSE);
			END_IF
			
			IF THIS^.fbStateMachineManual.StateComplete THEN
				THIS^.fbStateMachineManual.StateComplete		:=		FALSE;
			END_IF
			
		E_PMLState.RESETTING:
		
			IF NOT bResetIsSetToTrue THEN
				bResetIsSetToTrue		:=	TRUE;
				fbSeparatingModule.Reset(	bReset		:=		TRUE);
				fbMetalSortingModule.Reset(	bReset		:=		TRUE);
				fbPlasticSortingModule.Reset(bReset 	:=		TRUE);
			END_IF
				
			IF fbSeparatingModule.bState_ResetDone AND fbMetalSortingModule.bState_ResetDone AND fbPlasticSortingModule.bState_ResetDone AND
				fbSeparatingModule.bState_BarrierAtBasePos AND fbSeparatingModule.bState_ClampAtBasePos AND fbMetalSortingModule.bState_CylAtBasePos AND fbPlasticSortingModule.bState_CylAtBasePos THEN
					nBoxesOnTransport					:=	0;
					fbStateMachineMaintenance.StateComplete	:=	TRUE;
			END_IF
	END_CASE
END_METHOD

METHOD PRIVATE Operating_SemiAutomatic
VAR_INPUT
END_VAR

	CASE e_PMLState OF
		
		E_PMLState.IDLE:
			IF bResetIsSetToTrue THEN
				bResetIsSetToTrue		:=		FALSE;
				fbSeparatingModule.Reset(			bReset			:=	FALSE);
				fbMetalSortingModule.Reset(			bReset			:=	FALSE);
				fbPlasticSortingModule.Reset(		bReset			:=	FALSE);
				
				THIS^.fbStateMachineAuto.StateComplete				:=	FALSE;
			END_IF
		
		E_PMLState.STARTING:
			IF NOT bStartingIsSetToTrue THEN
				bStartingIsSetToTrue		:=		TRUE;
				fbSeparatingModule.Starting(		bStarting		:=	TRUE);
				fbMetalSortingModule.Starting(		bStarting		:=	TRUE);
				fbPlasticSortingModule.Starting(	bStarting		:=	TRUE);
			END_IF
			
			IF fbSeparatingModule.bState_StartingDone AND fbMetalSortingModule.bState_StartingDone AND fbPlasticSortingModule.bState_StartingDone THEN
				THIS^.fbStateMachineSemiAuto.StateComplete		:=		TRUE;
			END_IF
			
		E_PMLState.EXECUTE:
			IF bStartingIsSetToTrue	THEN
				bStartingIsSetToTrue		:=		FALSE;
				fbSeparatingModule.Starting(		bStarting		:=	FALSE);
				fbMetalSortingModule.Starting(		bStarting		:=	FALSE);
				fbPlasticSortingModule.Starting(	bStarting		:=	FALSE);
				
				THIS^.fbStateMachineAuto.StateComplete				:=	FALSE;
			END_IF
			
				fbSeparatingModule.Semiautomatic();
				fbMetalSortingModule.Semiautomatic();
				fbPlasticSortingModule.Semiautomatic();
				
			IF fbTriggerSeparated.Q THEN
				nBoxesOnTransport		:=		nBoxesOnTransport	+	1;
			END_IF
			
			IF fbTriggerMetalSorted	THEN
				nBoxesOnTransport		:=		nBoxesOnTransport	-	1;
			END_IF
			
			IF fbTriggerPlasticSorted THEN
				nBoxesOnTransport		:=		nBoxesOnTransport	-	1;
			END_IF
		
		E_PMLState.ABORTING:
			IF NOT bHaltIsSetToTrue THEN
				bHaltIsSetToTrue		:=		TRUE;
				fbSeparatingModule.Stop(			bStop			:=	TRUE);
				fbMetalSortingModule.Stop(			bStop			:=	TRUE);
				fbPlasticSortingModule.Stop(		bStop			:=	TRUE);
			END_IF
			
			IF fbSeparatingModule.bState_HaltDone AND fbMetalSortingModule.bState_HaltDone AND fbPlasticSortingModule.bState_HaltDone THEN
				THIS^.fbStateMachineSemiAuto.StateComplete			:=	TRUE;
			END_IF
			
		E_PMLState.ABORTED:
			IF bHaltIsSetToTrue THEN
				bHaltIsSetToTrue		:=		FALSE;
				fbSeparatingModule.Stop(			bStop			:=	FALSE);
				fbMetalSortingModule.Stop(			bStop			:=	FALSE);
				fbPlasticSortingModule.Stop(		bStop			:=	FALSE);
			END_IF
			
			IF THIS^.fbStateMachineSemiAuto.StateComplete THEN
				THIS^.fbStateMachineSemiAuto.StateComplete			:=	FALSE;
			END_IF
			
		E_PMLState.CLEARING:
			THIS^.fbStateMachineSemiAuto.StateComplete		:=	TRUE;
			
		E_PMLState.STOPPING:
			IF fbTriggerSeparated.Q THEN
				nBoxesOnTransport		:=		nBoxesOnTransport	+	1;
			END_IF
			
			IF fbTriggerMetalSorted	THEN
				nBoxesOnTransport		:=		nBoxesOnTransport	-	1;
			END_IF
			
			IF fbTriggerPlasticSorted THEN
				nBoxesOnTransport		:=		nBoxesOnTransport	-	1;
			END_IF
			
			IF nBoxesOnTransport = 0 AND NOT bHaltIsSetToTrue THEN
				bHaltIsSetToTrue		:=		TRUE;
				fbSeparatingModule.Stop(	bStop		:=		TRUE);
				fbMetalSortingModule.Stop(	bStop		:=		TRUE);
				fbPlasticSortingModule.Stop(bStop		:=		TRUE);
			END_IF
			
			IF fbSeparatingModule.bState_HaltDone AND fbMetalSortingModule.bState_HaltDone AND fbPlasticSortingModule.bState_HaltDone THEN
				THIS^.fbStateMachineSemiAuto.StateComplete			:=	TRUE;
			END_IF
		
		E_PMLState.STOPPED:
			IF bHaltIsSetToTrue THEN
				bHaltIsSetToTrue		:=		FALSE;
				fbSeparatingModule.Stop(			bStop			:=	FALSE);
				fbMetalSortingModule.Stop(			bStop			:=	FALSE);
				fbPlasticSortingModule.Stop(		bStop			:=	FALSE);
			END_IF
			
			IF THIS^.fbStateMachineSemiAuto.StateComplete THEN
				THIS^.fbStateMachineSemiAuto.StateComplete			:=	FALSE;
			END_IF
		
		E_PMLState.RESETTING:
			IF NOT bResetIsSetToTrue THEN
				bResetIsSetToTrue		:=		TRUE;
				fbSeparatingModule.Reset(	bReset		:=		TRUE);
				fbMetalSortingModule.Reset(	bReset		:=		TRUE);
				fbPlasticSortingModule.Reset(bReset 	:=		TRUE);
			END_IF
			
			IF fbSeparatingModule.bState_ResetDone AND fbMetalSortingModule.bState_ResetDone AND fbPlasticSortingModule.bState_StartingDone AND
				fbSeparatingModule.bState_BarrierAtBasePos AND fbSeparatingModule.bState_ClampAtBasePos AND
				fbMetalSortingModule.bState_CylAtBasePos AND fbPlasticSortingModule.bState_CylAtBasePos THEN
				nBoxesOnTransport							:=		0;
				THIS^.fbStateMachineSemiAuto.StateComplete	:=		TRUE;
			END_IF
	END_CASE
END_METHOD

END_FUNCTION_BLOCK

(* stored: Version 1.1.0.1, ProductVersion 3.1.4024.15
   POU FB_Machine: Id {7df4617e-7bb3-4f25-9837-0921844f24cd}, SpecialFunc None
   Method General_Enable: Id {149a393a-f524-48ce-8b52-2e7f8acc163e}
   Method General_Init: Id {55365572-5464-4324-b42a-b7f4ab586035}
   Method General_ModuleInputs: Id {e0890453-aacc-478b-ba67-4b9c253d8077}
   Method General_Requests: Id {8a9880e1-4cd2-48c8-a695-7a2a0f457a01}
   Method General_SetOutputs: Id {49d1f09e-8dc3-4742-bd71-b7e9ff71a432}
   Method General_StateMachine: Id {c0e031ad-ac3a-46a2-9330-e9ec0efefc5c}
   Method Operating_Automatic: Id {2aaebcd9-7bb6-42a0-9ada-aa72bc56fc0d}
   Method Operating_Maintenance: Id {06210250-0755-41fc-8866-aa6da8184b66}
   Method Operating_Manual: Id {eedf66c5-5d95-4d77-9169-88b2176b3cb4}
   Method Operating_SemiAutomatic: Id {2e013eba-aa9c-4402-a095-1c52f483942e} *)
